TYPE ST_Trackpads :
STRUCT
	One: ST_Trackpad;
	Two: ST_Trackpad;
END_STRUCT
END_TYPE

(* stored: Version 1.1.0.1
   DUT ST_Trackpads: Id {e4026d17-babf-4f21-9b81-8b66dca5d5cd} *)
